Universal Robots PolyScope program: taskboard_put_nut_tool_back.urp

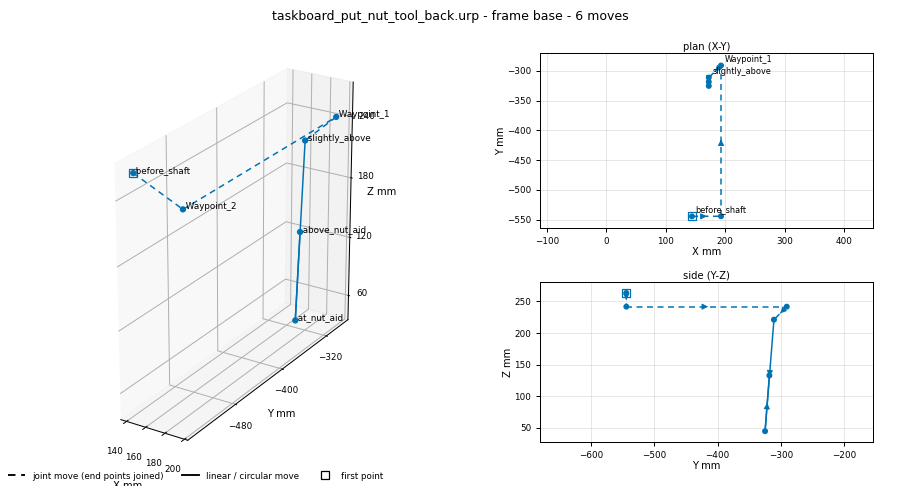
[picture p0: tool path of taskboard_put_nut_tool_back.urp in frame base, 6 of 6 moves have a stored position in this frame; points joined in program order, loops and branches not executed]
Program taskboard_put_nut_tool_back (installation=default directory=/programs/wrs2020 createdIn=5.6.0.90886 lastSavedIn=5.9.1.1031110 robotSerialNumber=20205500180)
Calibrated DH parameters: a=[0, -0.425, -0.3922, 0, 0, 0]; d=[0.1625, 0, 0, 0.1333, 0.0997, 0.0996]; alpha=[1.570796, 0, 0, 1.570796, -1.570796, 0]; deltaTheta=[0, 0, 0, 0, 0, 0]
Robot Program (runOnlyOnce=true)
  MoveJ speed 60 deg/s, acceleration 80 deg/s^2 (useActiveTCP=true) feature=Base
    Waypoint before_shaft: motionParameters(jointSpeed=1.047198 jointAcceleration=1.396263 cartesianSpeed=0.25 cartesianAcceleration=1.2); TCP in base x=144.251 y=-544.485 z=263.341 mm, rx=2.2425 ry=2.1895 rz=-0.0817 rad; joints [92.3, -83.868, 84.821, -93.226, -91.975, -266.37] deg; TCP offset x=0 y=0 z=220 mm, rx=0 ry=0 rz=0 rad
    Waypoint Waypoint_2: motionParameters(jointSpeed=2.094395 jointAcceleration=2.094395 cartesianSpeed=0.25 cartesianAcceleration=1.2 blendRadius=0.05); TCP in base x=193.098 y=-544.308 z=241.653 mm, rx=-2.26 ry=-2.0992 rz=0.0999 rad; joints [98.952, -79.277, 82.032, -92.106, -94.688, -256.794] deg
    Waypoint Waypoint_1: motionParameters(jointSpeed=2.094395 jointAcceleration=2.094395 cartesianSpeed=0.25 cartesianAcceleration=1.2 blendRadius=0.034); TCP in base x=193.098 y=-290.824 z=241.653 mm, rx=-2.26 ry=-2.0992 rz=0.0999 rad; joints [105.872, -111.142, 110.658, -88.291, -94.599, -249.911] deg
    Waypoint slightly_above: TCP in base x=172.519 y=-311.073 z=221.087 mm, rx=3.1334 ry=-0.0123 rz=-0.0179 rad; joints [97.806, -112.461, 114.667, -92.492, -90.559, -171.799] deg
  MoveL speed 250 mm/s, acceleration 1200 mm/s^2 (useActiveTCP=true) feature=Base
    Waypoint at_nut_aid: TCP in base x=172.519 y=-325.105 z=44.86 mm, rx=3.1334 ry=-0.0123 rz=-0.0179 rad; joints [97.451, -101.585, 134.781, -123.486, -90.53, -172.054] deg
    URCap Gripper (Robotiq_Grippers, Robotiq Inc.) dataModel(position=21.96078431372549, force=100.0, speed=100.0, positionInDouble=21.96078431372549, forceInDouble=100.0, speedInDouble=100.0, slaveIds=[9], blocking=true)
    Waypoint above_nut_aid: TCP in base x=172.519 y=-318.273 z=132.878 mm, rx=3.1334 ry=-0.0123 rz=-0.0179 rad; joints [97.626, -109.17, 125.745, -106.863, -90.541, -171.937] deg
